FUNCTION_BLOCK data2event (* Service Interface Function Block Type *)
  (* Standard: 61499-2 *)
  (* Version 0.1, 2017-03-03, WD, YY Automation *)
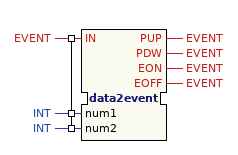
  EVENT_INPUT
    IN : EVENT WITH num1, num2; (* Service Initialization *)
  END_EVENT
  EVENT_OUTPUT
    PUP : EVENT; (* Initialization Confirm *)
    PDW : EVENT;
    EON : EVENT;
    EOFF : EVENT;
  END_EVENT
  VAR_INPUT
    num1 : INT; (* Event Input Qualifier *)
    num2 : INT;
  END_VAR
END_FUNCTION_BLOCK
(* other elements stored in the file *)
(* VarDeclaration Name=state Type=BOOL *)
(* Algorithm Name=exchange *)
(* Other Language=CPP Text=if( num1==num2){ fbptr->emitEO("EON"); if(!state){ fbptr->emitEO("PUP"); state=true; } } else{ if(state){ fbptr->emitEO("PDW"); } fbptr->emitEO("EOFF"); } *)
